(* IEC 61131-3 sources: SJ_AGV/PLC/Standard_functions.4.4.0/SubFunctions, 7 files *)

(* ---- BytesToInt_FB.ST ---- *)
FUNCTION_BLOCK BytesToInt_FB
VAR_EXTERNAL
	NDC8:NDC8_T;
	MegaWord:word;
	HighByte:byte;
	LowByte:byte;
END_VAR

VAR_INPUT
	Byte1 : byte;
	Byte2 : byte;
END_VAR

VAR_OUTPUT
	IntValue : int;
END_VAR

VAR
	littleEndian:bool := true;
END_VAR
(*
 -----------------------------------------------------------------------------------
 BytesToInt_FB
 -----------------------------------------------------------------------------------

 Description:
 Combines two bytes to an INT.
 littleEndian is used to control if least or most significant byte should come first.

 Rev 	Who		Date  		Desc
 -----------------------------------------------------------------------------------
 0.1  	KJN  	140206		Created
 -----------------------------------------------------------------------------------*)

if littleEndian then	(* First byte is least significant *)

	LowByte := Byte2;
	HighByte := Byte1;

	IntValue := word_to_int(MegaWord);

else					(* Second byte is least significant *)

	LowByte := Byte1;
	HighByte := Byte2;

	IntValue := word_to_int(MegaWord);

end_if;
END_FUNCTION_BLOCK

(* ---- BytesToUInt_FB.ST ---- *)
FUNCTION_BLOCK BytesToUInt_FB
VAR_EXTERNAL
	NDC8:NDC8_T;
	MegaWord:word;
	HighByte:byte;
	LowByte:byte;

END_VAR

VAR_INPUT
	Byte1 : byte;
	Byte2 : byte;
END_VAR

VAR_OUTPUT
	UIntValue : uint;
END_VAR

VAR
	littleEndian:bool := true;
END_VAR
(*
 -----------------------------------------------------------------------------------
 BytesToInt_FB
 -----------------------------------------------------------------------------------

 Description:
 Combines two bytes to an UINT.
 littleEndian is used to control if least or most significant byte should come first.

 Rev 	Who		Date  		Desc
 -----------------------------------------------------------------------------------
 0.1  	KJN  	140206		Created
 -----------------------------------------------------------------------------------*)

if littleEndian then	(* First byte is least significant *)

	LowByte := Byte2;
	HighByte := Byte1;

	UIntValue := word_to_uint(MegaWord);

else					(* Second byte is least significant *)

	LowByte := Byte1;
	HighByte := Byte2;

	UIntValue := word_to_uint(MegaWord);

end_if;
END_FUNCTION_BLOCK

(* ---- DateAndTime_FB.ST ---- *)
FUNCTION_BLOCK DateAndTime_FB
VAR_EXTERNAL
	NDC8:NDC8_T;

END_VAR

VAR_INPUT
	UTC_Clock	:	DINT;
END_VAR

VAR_OUTPUT
	ErrorCode	:	DINT;	(* 	0 = No errors
								1 = No UTC time input *)

	Year,Month,Day	:	DINT;
	Hours,Minutes,Seconds	:	DINT;
	DayWeek			:	STRING;

END_VAR

VAR
	Curr_Year, Temp_Days,Rem_Days	:	DINT;
	Rem_Seconds,Temp_Seconds	:	DINT;
	Days		:	DINT;
	Years_Bi	:	ARRAY [1..18] of DINT := [1972,1976,1980,1984,1988,1992,1996,2000,2004,2008,2012,2016,2020,2024,2028,2032,2036,2040];
	Months		:	ARRAY [1..12] of DINT := [31,28,31,30,31,30,31,31,30,31,30,31];
	WeekDays	:	ARRAY [0..6] of STRING := ['Thursday','Friday','Saturday','Sunday','Monday','Tuesday','Wednesday'];
	Start_Year 	: 	DINT := 1970;
	j,i,k		:	DINT := 1;
	Bissextile	:	BOOL;
END_VAR
(* Calculate date and time from UTC Clock NDC8.Vmc.Clock
-------------------------------------------
Seconds since 00:00:00 (Thursday) January 1 1970.
Valid after the vehicle controller has connected to System Manager
followed by a restart of the vehicle controller. *)

If UTC_Clock < 0 then
	ErrorCode := 1;
	Return;			(* Error, exit from FB *)
End_If;

(* How many days since 00:00:00 January 1 1970 *)
Days := UTC_Clock / (60*60*24);

(* Remaining seconds from days *)
Rem_Seconds := UTC_Clock - (Days*60*60*24);

(* Day of week *)
k := Days mod 7;
k := LIMIT(0,k,6);
DayWeek := WeekDays[k];	(* Week day *)

(* Init *)
Curr_Year := Start_Year;
Temp_Days := Days;
Temp_Seconds := Rem_Seconds;
j := 1;
i := 1;

(* Year *)
while Temp_Days > 364 do
	if Years_Bi[j] = Curr_Year then
		Temp_Days := Temp_Days - 366;
		j := j+1;
		j := LIMIT(1,j,18);
	else
		Temp_Days := Temp_Days - 365;
	end_if;
	Rem_Days := Temp_Days + 1;	(* 1 day gone means January 2th so we need to add 1 day *)
	Curr_Year := Curr_Year + 1;
	Year := Curr_Year;			(* Year *)
end_while;

(* Bissextile? *)
for j := 1 to 12 do
	if Year = Years_Bi[j] then
		Bissextile := true;
		exit;		(* exit if Bissextile *)
	else
		Bissextile := false;
	end_if;
end_for;

(* Month *)
If 	Rem_Days < 28 then
	Month := i;				(* Month *)
	Day := Rem_Days;		(* Day *)
else

	while Rem_Days > 27 do
		If i = 2 then	(* February? *)
			if Bissextile then
				Rem_Days := Rem_Days - Months[i] - 1;	(* 29 days for Bissextile year *)
			else
				Rem_Days := Rem_Days - Months[i];
			end_if;
		else
			Rem_Days := Rem_Days - Months[i];
		end_if;
		i := i + 1;
		i := LIMIT(1,i,12);
		Month := i;				(* Month *)
		Day := Rem_Days;		(* Day *)
	end_while;
end_if;

(* Hours *)
Hours := Temp_Seconds / 3600;
Temp_Seconds := Rem_Seconds - (Hours*3600);

(* Minutes *)
Minutes := Temp_Seconds / 60;

(* Seconds *)
Seconds := Rem_Seconds - (Hours*3600) - (Minutes*60);

ErrorCode := 0;		(* No errors *)

END_FUNCTION_BLOCK

(* ---- FourBytesToUDInt_FB.ST ---- *)
FUNCTION_BLOCK FourBytesToUDInt_FB
VAR_EXTERNAL
	NDC8:NDC8_T;
	DMegaWord:dword;
	FirstByte:byte;
	SecondByte:byte;
	ThirdByte:byte;
	FourthByte:byte;

END_VAR

VAR_INPUT
	Byte1 : byte;
	Byte2 : byte;
	Byte3 : byte;
	Byte4 : byte;
END_VAR

VAR_OUTPUT
	UDIntValue : udint;
END_VAR

VAR
	littleEndian:bool := true;
END_VAR
(*
 -----------------------------------------------------------------------------------
 FourBytesToUDInt_FB
 -----------------------------------------------------------------------------------

 Description:
 Combines two bytes to an UINT.
 littleEndian is used to control if least or most significant byte should come first.

 Rev 	Who		Date  		Desc
 -----------------------------------------------------------------------------------
 0.1  	KJN  	140206		Created
 -----------------------------------------------------------------------------------*)

if littleEndian then	(* First byte is least significant *)

	FirstByte	:= Byte1;
	SecondByte	:= Byte2;
	ThirdByte	:= Byte3;
	FourthByte	:= Byte4;

	UDIntValue := dword_to_udint(DMegaWord);
else					(* Second byte is least significant *)

	FirstByte	:= Byte3;
	SecondByte	:= Byte4;
	ThirdByte	:= Byte1;
	FourthByte	:= Byte2;

	UDIntValue := dword_to_udint(DMegaWord);

end_if;
END_FUNCTION_BLOCK

(* ---- IntToByteArray_FB.ST ---- *)
FUNCTION_BLOCK IntToByteArray_FB
VAR_EXTERNAL
	NDC8:NDC8_T;
	MegaWord:word;
	HighByte:byte;
	LowByte:byte;
END_VAR

VAR_INPUT
	IntValue : int;
END_VAR

VAR_OUTPUT
	ByteArray : ARRAY[1..2] OF BYTE;
END_VAR

VAR
	littleEndian:bool := true;
END_VAR
(*
 -----------------------------------------------------------------------------------
 IntToByteArray_FB
 -----------------------------------------------------------------------------------

 Description:
 Splits INT into an array of two bytes.
 littleEndian is used to control if least or most significant byte should come first.

 Rev 	Who		Date  		Desc
 -----------------------------------------------------------------------------------
 0.1  	KJN  	140205		Created
 -----------------------------------------------------------------------------------*)

(* Get word. Saved at same data positions as HighByte and LowByte *)
MegaWord := int_to_word(IntValue);

if littleEndian then	(* Start with least significant byte *)

	ByteArray[1] := HighByte;
	ByteArray[2] := LowByte;

else				(* Start with most significant byte *)

	ByteArray[2] := HighByte;
	ByteArray[1] := LowByte;

end_if;
END_FUNCTION_BLOCK

(* ---- SENSORHANDLING_FB.ST ---- *)
FUNCTION_BLOCK SENSORHANDLING_FB
VAR_EXTERNAL

END_VAR

VAR_INPUT
	Input		: bool;
	EventID		: dint;
	StopStringID: dint;
	Enable		: bool;
	OnDelay		: time;
	OffDelay 	: time;
END_VAR

VAR_OUTPUT
	Stop	: bool;
END_VAR

VAR
	OnFilterTON	: TON;
	OffFilterTP: TP;
	StopRT		: R_Trig;
	Off_FT		: F_Trig;
END_VAR
(* filter indata with on delay *)
OnFilterTON(IN:=Input, PT:=OnDelay);

(* Off delay *)
OffFilterTP(IN:=OnFilterTON.q, PT:=OffDelay);

(* Set/reset or disable stop signal. *)
if not Enable then
	Stop:=false;
elsif OnFilterTON.Q then
	Stop:=true;
elsif not OffFilterTP.q then
	Stop:=false;
end_if;

(* generate events *)
StopRT(CLK:=Stop);
if StopRT.Q then
	;
end_if;

(* Display update *)
DisplayStopString(INStatus:=Stop, StopString:=StopStringID, StopValue:=0);

END_FUNCTION_BLOCK

(* ---- UIntToByteArray_FB.ST ---- *)
FUNCTION_BLOCK UIntToByteArray_FB
VAR_EXTERNAL
	NDC8:NDC8_T;
	MegaWord:word;
	HighByte:byte;
	LowByte:byte;
END_VAR

VAR_INPUT
	UIntValue : uint;
END_VAR

VAR_OUTPUT
	ByteArray : ARRAY[1..2] OF BYTE;
END_VAR

VAR
	shift:shl_word;
	littleEndian:bool := true;
	tempWord:word;

END_VAR
;

(*
 -----------------------------------------------------------------------------------
 IntToByteArray_FB
 -----------------------------------------------------------------------------------

 Description:
 Splits UINT into an array of two bytes.
 littleEndian is used to control if least or most significant byte should come first.

 Rev 	Who		Date  		Desc
 -----------------------------------------------------------------------------------
 0.1  	KJN  	140205		Created
 -----------------------------------------------------------------------------------*)

(* Get word. Saved at same data positions as HighByte and LowByte *)
MegaWord := uint_to_word(UIntValue);

if littleEndian then	(* Start with least significant byte *)

	ByteArray[1] := HighByte;
	ByteArray[2] := LowByte;

else					(* Start with most significant byte *)

	ByteArray[2] := HighByte;
	ByteArray[1] := LowByte;

end_if;
END_FUNCTION_BLOCK
